// TIA Portal V20 export
TYPE "LKinCtrl_PathEditor_typeCommandEditorExternalEvents"
// stored: Access Published
   STRUCT
      setContent { ExternalAccessible := 'False'; ExternalVisible := 'False'; ExternalWritable := 'False'} : Struct
         trigger : Bool;   // triggers internal event. Reset internally.
         contentType : Int;   // 10: variables, 11: conditions, 12: Inputs, 13: Outputs, 14: Points, 20: Axes, 21: PosSyncAxes , 22: SyncAxes, 30: Labels, 40: Sequences
      END_STRUCT;
      changeSelection { ExternalAccessible := 'False'; ExternalVisible := 'False'; ExternalWritable := 'False'} : Struct
         trigger : Bool;   // triggers event. Reset internally.
         noSelection : Bool := true;   // TRUE: nothing is selected in table.
         selectedIndex : DInt := -1;   // Selected index in table. Only valid if noSelection = FALSE.
      END_STRUCT;
      focusSelection { ExternalAccessible := 'False'; ExternalVisible := 'False'; ExternalWritable := 'False'} : Struct
         trigger : Bool;   // triggers internal event. Reset internally.
         selectedField : Int;   // field where selected index should be placed. Starting at 1.
      END_STRUCT;
      changeCommand { ExternalAccessible := 'False'; ExternalVisible := 'False'; ExternalWritable := 'False'} : Struct
         trigger : Bool;
         command : "LKinCtrl_typePathDataElement";
      END_STRUCT;
   END_STRUCT;
END_TYPE
